(* PLC project Generated.project, CODESYS CODESYS V3.5 SP19 Patch 1 *)
(* stored: creationDateTime 2026-09-01T01:00:08.916521, modificationDateTime 2026-09-01T01:00:08.916521 *)

(* ═══════════════════════════════════════════════════════════════ ⚙️ ST_CycleDumpAtTremieCfg — Réglages persistants cycle vidage trémie (legacy) ═══════════════════════════════════════════════════════════════ *)
TYPE ST_CycleDumpAtTremieCfg : STRUCT
  Initialized : BOOL := FALSE;  (* 🚦 flag restauration boot *)
END_STRUCT;
END_TYPE
